// TIA Portal project "Project_Metrou" (V15.1)

(* hardware
DEVICE "S71500/ET200MP station_1"  S7-1500 station
   slot 0: "Rail_0"  Rack  6ES7 590-1***0-0AA0
   slot 1: "PLC_1"  CPU 1513-1 PN  6ES7 513-1AL02-0AB0  V2.6
      slot 3: "CPU display_1"  6ES7591-1AA00-0AA0
*)

// ===== PLC "PLC_1"  CPU 1513-1 PN =====

DATA_BLOCK "Alarme_scara"   // DB1
{ S7_Optimized_Access := 'TRUE' }
VERSION : 0.1
   VAR
      alarme_gather : Word;
      alarme_vect : Array[0..15] of Bool;
   END_VAR
BEGIN
END_DATA_BLOCK

DATA_BLOCK "Avarii"   // DB2
{ S7_Optimized_Access := 'TRUE' }
VERSION : 0.1
   VAR
      esd : Bool;
      esd_btn : Bool;
      reset_esd : Bool;
      avarie_s1 : Bool;
      avarie_s2 : Bool;
      reset_avarii : Bool;
   END_VAR
BEGIN
END_DATA_BLOCK

DATA_BLOCK "Alarme_poarta"   // DB3
{ S7_Optimized_Access := 'TRUE' }
VERSION : 0.1
   VAR
      alarme_gather : Word;
      alarme_vect : Array[0..15] of Bool;
   END_VAR
BEGIN
END_DATA_BLOCK

DATA_BLOCK "Scara1_DB"   // DB4
{ S7_Optimized_Access := 'TRUE' }
VERSION : 0.1
// stored: InstanceOfName Scara
"Scara"
BEGIN
END_DATA_BLOCK

DATA_BLOCK "Scara2_DB"   // DB5
{ S7_Optimized_Access := 'TRUE' }
VERSION : 0.1
// stored: InstanceOfName Scara
"Scara"
BEGIN
END_DATA_BLOCK

DATA_BLOCK "Variabile_scara1"   // DB6
{ S7_Optimized_Access := 'TRUE' }
VERSION : 0.1
   VAR
      curent_stea : Real;
      curent_triunghi : Real;
      senzor_presiune : Bool;
      porniire_stea : Bool;
      pornire_triunghi : Bool;
      start : Bool;
      stop : Bool;
      directie : Bool;
      directie_sus : Bool;
      directie_jos : Bool;
      reseteaza_directia : Bool;
   END_VAR
BEGIN
END_DATA_BLOCK

DATA_BLOCK "Variabile_scara2"   // DB7
{ S7_Optimized_Access := 'TRUE' }
VERSION : 0.1
   VAR
      curent_stea : Real;
      curent_triunghi : Real;
      senzor_presiune : Bool;
      porniire_stea : Bool;
      pornire_triunghi : Bool;
      start : Bool;
      stop : Bool;
      directie : Bool;
      directie_sus : Bool;
      directie_jos : Bool;
      reseteaza_directia : Bool;
   END_VAR
BEGIN
END_DATA_BLOCK

// folder: System blocks/Program resources

DATA_BLOCK "reset_esd"   // DB8
{ S7_Optimized_Access := 'TRUE' }
AUTHOR : Simatic
FAMILY : IEC
NAME : IEC_TMR
VERSION : 1.0
// stored: InstanceOfName IEC_TIMER
"IEC_TIMER"
BEGIN
END_DATA_BLOCK

// folder: (top level)

FUNCTION_BLOCK "Scara"   // FB1, LAD
{ S7_Optimized_Access := 'TRUE' }
VERSION : 0.1
   VAR_INPUT
      esd : Bool;
      curent_stea : Real;
      curent_triunghi : Real;
      senzor_presiune : Bool;
      avarie_scara : Bool;
   END_VAR
   VAR_OUTPUT
      stea : Bool;
      triunghi : Bool;
      directie_selectata : Bool;
   END_VAR
   VAR_IN_OUT
      reseteaza_directia : Bool;
      stop : Bool;
      start : Bool;
      directie_sus : Bool;
      directie_jos : Bool;
   END_VAR
   VAR
      pornire_stea : Bool;
      pornire_triunghi : Bool;
      permisiune_pornire : Bool;
      permisie_repornire : Bool;
      timer_stop : TON_TIME;
      Motor : "Motor";
   END_VAR
BEGIN

REGION Network 1: da permisiuneade pornire la scara
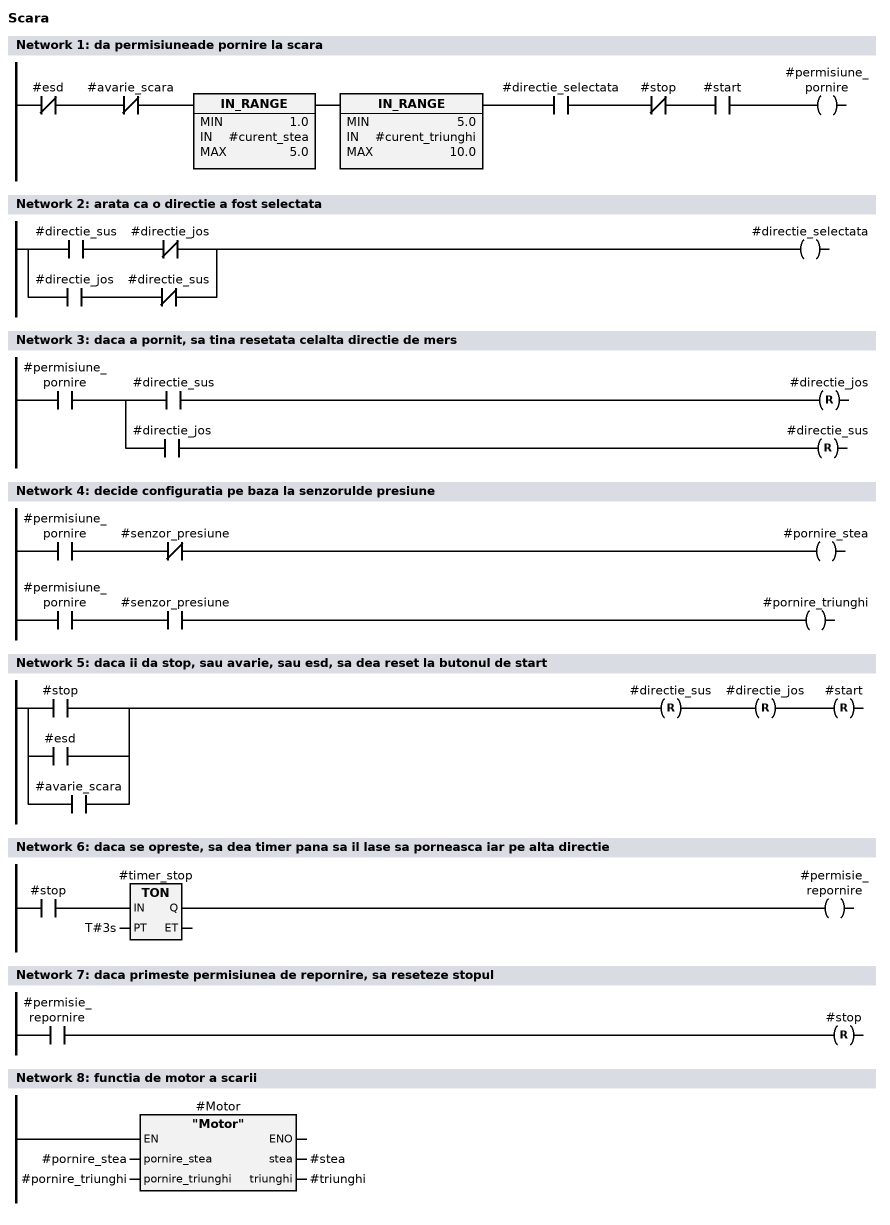
   RUNG wire#powerrail
      I_Contact( #esd )
      I_Contact( #avarie_scara )
      { S7_Templates := "SrcType := Real" } InRange(min := 1.0, in := #curent_stea, max := 5.0)
      { S7_Templates := "SrcType := Real" } InRange(min := 5.0, in := #curent_triunghi, max := 10.0)
      Contact( #directie_selectata )
      I_Contact( #stop )
      Contact( #start )
      Coil( #permisiune_pornire )
   END_RUNG
   // the same network as SCL:
   #permisiune_pornire := NOT #esd AND NOT #avarie_scara AND (1.0 <= #curent_stea) AND (#curent_stea <= 5.0) AND (5.0 <= #curent_triunghi) AND (#curent_triunghi <= 10.0) AND #directie_selectata AND NOT #stop AND #start;
END_REGION

REGION Network 2: arata ca o directie a fost selectata
   RUNG wire#powerrail
      Contact( #directie_sus )
      I_Contact( #directie_jos )
      wire#w1
      Coil( #directie_selectata )
   END_RUNG
   RUNG wire#powerrail
      Contact( #directie_jos )
      I_Contact( #directie_sus )
   END_RUNG wire#w1
   // the same network as SCL:
   #directie_selectata := (#directie_sus AND NOT #directie_jos) OR (#directie_jos AND NOT #directie_sus);
END_REGION

REGION Network 3: daca a pornit, sa tina resetata celalta directie de mers
   RUNG wire#powerrail
      Contact( #permisiune_pornire )
      wire#w1
      Contact( #directie_sus )
      R_Coil( #directie_jos )
   END_RUNG
   RUNG wire#w1
      Contact( #directie_jos )
      R_Coil( #directie_sus )
   END_RUNG
   // the same network as SCL:
   IF #permisiune_pornire AND #directie_sus THEN #directie_jos := FALSE; END_IF;
   IF #permisiune_pornire AND #directie_jos THEN #directie_sus := FALSE; END_IF;
END_REGION

REGION Network 4: decide configuratia pe baza la senzorulde presiune
   RUNG wire#powerrail
      Contact( #permisiune_pornire )
      I_Contact( #senzor_presiune )
      Coil( #pornire_stea )
   END_RUNG
   RUNG wire#powerrail
      Contact( #permisiune_pornire )
      Contact( #senzor_presiune )
      Coil( #pornire_triunghi )
   END_RUNG
   // the same network as SCL:
   #pornire_stea := #permisiune_pornire AND NOT #senzor_presiune;
   #pornire_triunghi := #permisiune_pornire AND #senzor_presiune;
END_REGION

REGION Network 5: daca ii da stop, sau avarie, sau esd, sa dea reset la butonul de start
   RUNG wire#powerrail
      Contact( #stop )
      wire#w1
      R_Coil( #directie_sus )
      R_Coil( #directie_jos )
      R_Coil( #start )
   END_RUNG
   RUNG wire#powerrail
      Contact( #esd )
   END_RUNG wire#w1
   RUNG wire#powerrail
      Contact( #avarie_scara )
   END_RUNG wire#w1
   // the same network as SCL:
   IF #stop OR #esd OR #avarie_scara THEN
       #directie_sus := FALSE;
       #directie_jos := FALSE;
       #start := FALSE;
   END_IF;
END_REGION

REGION Network 6: daca se opreste, sa dea timer pana sa il lase sa porneasca iar pe alta directie
   #timer_stop(IN := #stop, PT := T#3s);   // TON
   #permisie_repornire := #timer_stop.Q;
END_REGION

REGION Network 7: daca primeste permisiunea de repornire, sa reseteze stopul
   RUNG wire#powerrail
      Contact( #permisie_repornire )
      R_Coil( #stop )
   END_RUNG
   // the same network as SCL:
   IF #permisie_repornire THEN #stop := FALSE; END_IF;
END_REGION

REGION Network 8: functia de motor a scarii
   RUNG wire#powerrail
      #Motor(pornire_stea := #pornire_stea, pornire_triunghi := #pornire_triunghi, stea => #stea, triunghi => #triunghi)
   END_RUNG
   // the same network as SCL:
   #Motor(pornire_stea := #pornire_stea,   // "Motor"
          pornire_triunghi := #pornire_triunghi,
          stea => #stea,
          triunghi => #triunghi);
END_REGION
END_FUNCTION_BLOCK

FUNCTION_BLOCK "Motor"   // FB2, LAD
{ S7_Optimized_Access := 'TRUE' }
VERSION : 0.1
   VAR_INPUT
      pornire_stea : Bool;
      pornire_triunghi : Bool;
   END_VAR
   VAR_OUTPUT
      stea : Bool;
      triunghi : Bool;
   END_VAR
BEGIN

REGION Network 1: daca primeste plecare pe stea, sa o activeze
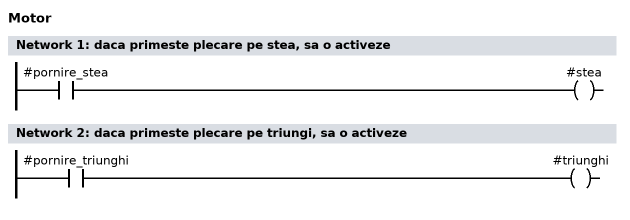
   RUNG wire#powerrail
      Contact( #pornire_stea )
      Coil( #stea )
   END_RUNG
   // the same network as SCL:
   #stea := #pornire_stea;
END_REGION

REGION Network 2: daca primeste plecare pe triungi, sa o activeze
   RUNG wire#powerrail
      Contact( #pornire_triunghi )
      Coil( #triunghi )
   END_RUNG
   // the same network as SCL:
   #triunghi := #pornire_triunghi;
END_REGION
END_FUNCTION_BLOCK

ORGANIZATION_BLOCK "Main"   // OB1, LAD, ProgramCycle
TITLE = "Main Program Sweep (Cycle)"
{ S7_Optimized_Access := 'TRUE' }
VERSION : 0.1
   VAR_INPUT
      Initial_Call : Bool;   // Initial call of this OB
      Remanence : Bool;   // =True, if remanent data are available
   END_VAR
   VAR_TEMP   // added for the SCL form of the ladder/FBD networks
      _w1 : Bool;
      _w2 : Bool;
      _w3 : Bool;
      _w4 : Bool;
      _w5 : Bool;
      _w6 : Bool;
   END_VAR
BEGIN

REGION Network 1: scara 1
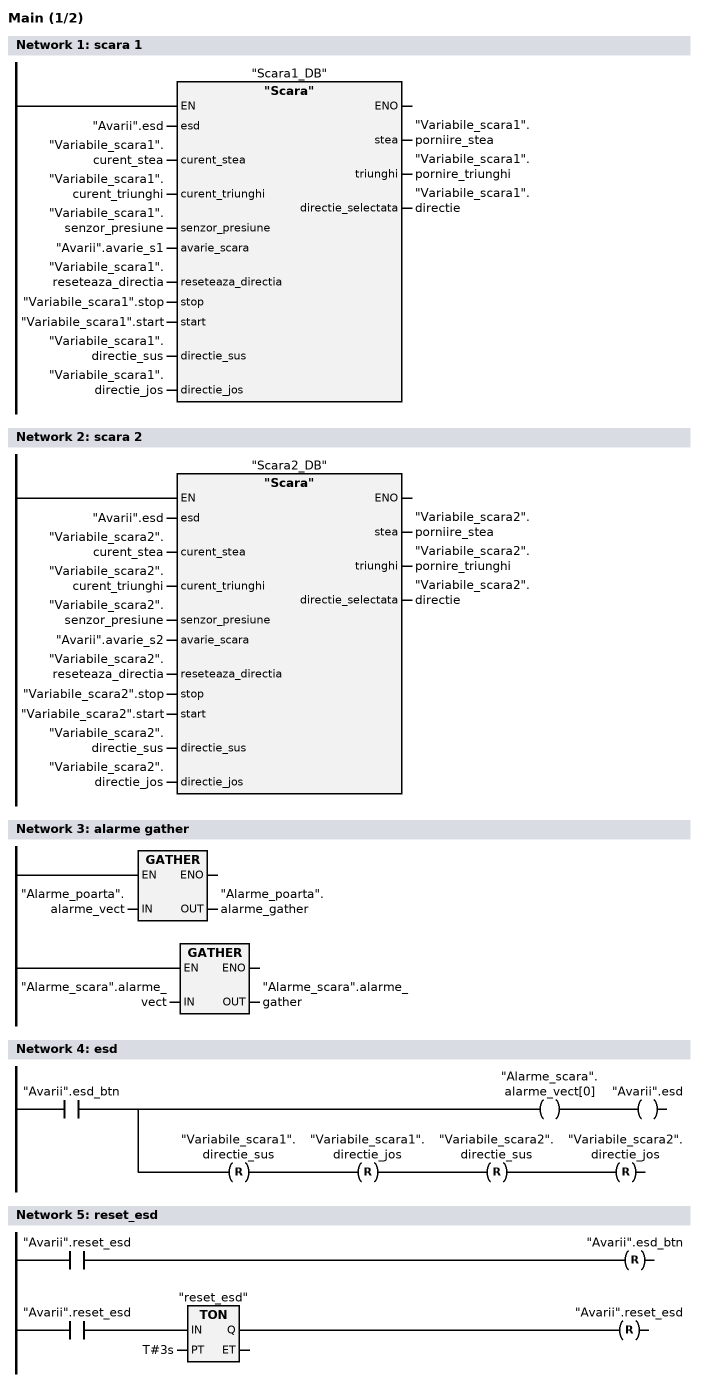
   RUNG wire#powerrail
      "Scara1_DB"(esd := "Avarii".esd, curent_stea := "Variabile_scara1".curent_stea, curent_triunghi := "Variabile_scara1".curent_triunghi, senzor_presiune := "Variabile_scara1".senzor_presiune, avarie_scara := "Avarii".avarie_s1, reseteaza_directia := "Variabile_scara1".reseteaza_directia, stop := "Variabile_scara1".stop, start := "Variabile_scara1".start, directie_sus := "Variabile_scara1".directie_sus, directie_jos := "Variabile_scara1".directie_jos, stea => "Variabile_scara1".porniire_stea, triunghi => "Variabile_scara1".pornire_triunghi, directie_selectata => "Variabile_scara1".directie)
   END_RUNG
   // the same network as SCL:
   "Scara1_DB"(esd := "Avarii".esd,   // "Scara"
               curent_stea := "Variabile_scara1".curent_stea,
               curent_triunghi := "Variabile_scara1".curent_triunghi,
               senzor_presiune := "Variabile_scara1".senzor_presiune,
               avarie_scara := "Avarii".avarie_s1,
               reseteaza_directia := "Variabile_scara1".reseteaza_directia,
               stop := "Variabile_scara1".stop,
               start := "Variabile_scara1".start,
               directie_sus := "Variabile_scara1".directie_sus,
               directie_jos := "Variabile_scara1".directie_jos,
               stea => "Variabile_scara1".porniire_stea,
               triunghi => "Variabile_scara1".pornire_triunghi,
               directie_selectata => "Variabile_scara1".directie);
END_REGION

REGION Network 2: scara 2
   RUNG wire#powerrail
      "Scara2_DB"(esd := "Avarii".esd, curent_stea := "Variabile_scara2".curent_stea, curent_triunghi := "Variabile_scara2".curent_triunghi, senzor_presiune := "Variabile_scara2".senzor_presiune, avarie_scara := "Avarii".avarie_s2, reseteaza_directia := "Variabile_scara2".reseteaza_directia, stop := "Variabile_scara2".stop, start := "Variabile_scara2".start, directie_sus := "Variabile_scara2".directie_sus, directie_jos := "Variabile_scara2".directie_jos, stea => "Variabile_scara2".porniire_stea, triunghi => "Variabile_scara2".pornire_triunghi, directie_selectata => "Variabile_scara2".directie)
   END_RUNG
   // the same network as SCL:
   "Scara2_DB"(esd := "Avarii".esd,   // "Scara"
               curent_stea := "Variabile_scara2".curent_stea,
               curent_triunghi := "Variabile_scara2".curent_triunghi,
               senzor_presiune := "Variabile_scara2".senzor_presiune,
               avarie_scara := "Avarii".avarie_s2,
               reseteaza_directia := "Variabile_scara2".reseteaza_directia,
               stop := "Variabile_scara2".stop,
               start := "Variabile_scara2".start,
               directie_sus := "Variabile_scara2".directie_sus,
               directie_jos := "Variabile_scara2".directie_jos,
               stea => "Variabile_scara2".porniire_stea,
               triunghi => "Variabile_scara2".pornire_triunghi,
               directie_selectata => "Variabile_scara2".directie);
END_REGION

REGION Network 3: alarme gather
   GATHER(IN := "Alarme_poarta".alarme_vect, OUT => "Alarme_poarta".alarme_gather);
   GATHER(IN := "Alarme_scara".alarme_vect, OUT => "Alarme_scara".alarme_gather);
END_REGION

REGION Network 4: esd
   RUNG wire#powerrail
      Contact( "Avarii".esd_btn )
      wire#w1
      Coil( "Alarme_scara".alarme_vect[0] )
      Coil( "Avarii".esd )
   END_RUNG
   RUNG wire#w1
      R_Coil( "Variabile_scara1".directie_sus )
      R_Coil( "Variabile_scara1".directie_jos )
      R_Coil( "Variabile_scara2".directie_sus )
      R_Coil( "Variabile_scara2".directie_jos )
   END_RUNG
   // the same network as SCL:
   "Alarme_scara".alarme_vect[0] := "Avarii".esd_btn;
   "Avarii".esd := "Avarii".esd_btn;
   IF "Avarii".esd_btn THEN
       "Variabile_scara1".directie_sus := FALSE;
       "Variabile_scara1".directie_jos := FALSE;
       "Variabile_scara2".directie_sus := FALSE;
       "Variabile_scara2".directie_jos := FALSE;
   END_IF;
END_REGION

REGION Network 5: reset_esd
   IF "Avarii".reset_esd THEN "Avarii".esd_btn := FALSE; END_IF;
   "reset_esd".TON(IN := "Avarii".reset_esd, PT := T#3s);
   IF "reset_esd".Q THEN "Avarii".reset_esd := FALSE; END_IF;
END_REGION

REGION Network 6: avarii pe scari, cu alarme pt hmi
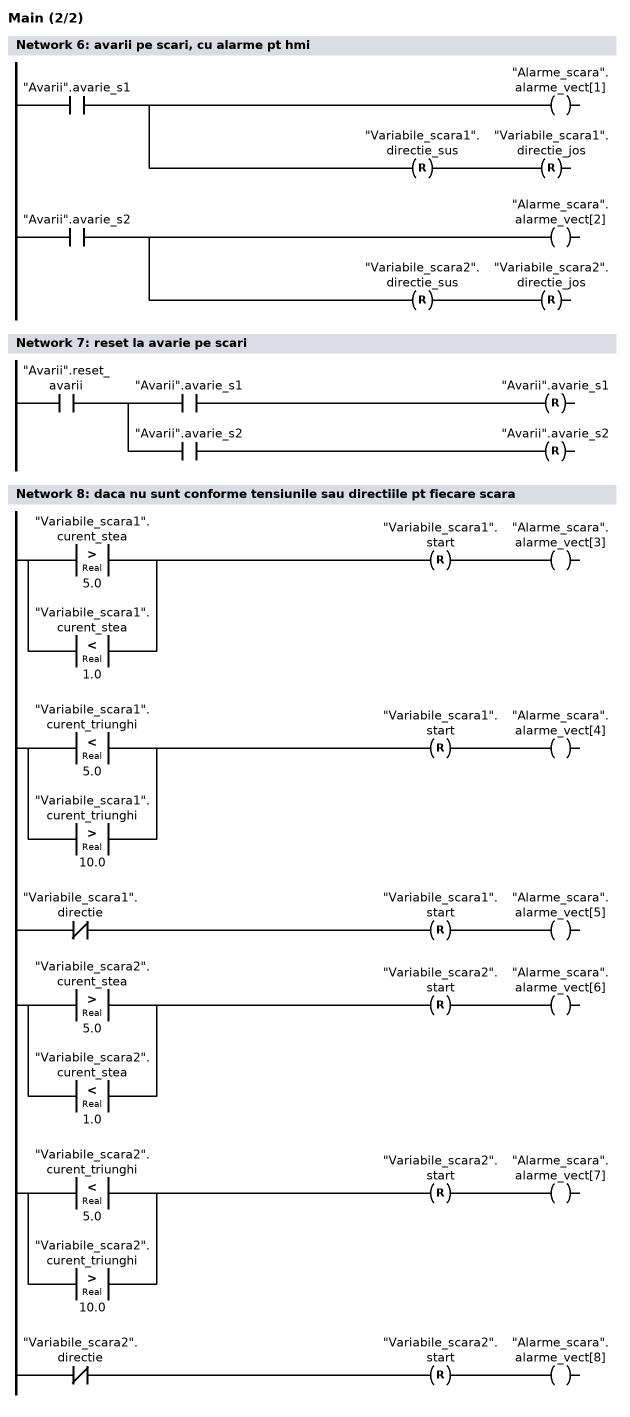
   RUNG wire#powerrail
      Contact( "Avarii".avarie_s1 )
      wire#w1
      Coil( "Alarme_scara".alarme_vect[1] )
   END_RUNG
   RUNG wire#w1
      R_Coil( "Variabile_scara1".directie_sus )
      R_Coil( "Variabile_scara1".directie_jos )
   END_RUNG
   RUNG wire#powerrail
      Contact( "Avarii".avarie_s2 )
      wire#w2
      Coil( "Alarme_scara".alarme_vect[2] )
   END_RUNG
   RUNG wire#w2
      R_Coil( "Variabile_scara2".directie_sus )
      R_Coil( "Variabile_scara2".directie_jos )
   END_RUNG
   // the same network as SCL:
   "Alarme_scara".alarme_vect[1] := "Avarii".avarie_s1;
   IF "Avarii".avarie_s1 THEN
       "Variabile_scara1".directie_sus := FALSE;
       "Variabile_scara1".directie_jos := FALSE;
   END_IF;
   "Alarme_scara".alarme_vect[2] := "Avarii".avarie_s2;
   IF "Avarii".avarie_s2 THEN
       "Variabile_scara2".directie_sus := FALSE;
       "Variabile_scara2".directie_jos := FALSE;
   END_IF;
END_REGION

REGION Network 7: reset la avarie pe scari
   RUNG wire#powerrail
      Contact( "Avarii".reset_avarii )
      wire#w1
      Contact( "Avarii".avarie_s1 )
      R_Coil( "Avarii".avarie_s1 )
   END_RUNG
   RUNG wire#w1
      Contact( "Avarii".avarie_s2 )
      R_Coil( "Avarii".avarie_s2 )
   END_RUNG
   // the same network as SCL:
   IF "Avarii".reset_avarii AND "Avarii".avarie_s1 THEN "Avarii".avarie_s1 := FALSE; END_IF;
   IF "Avarii".reset_avarii AND "Avarii".avarie_s2 THEN "Avarii".avarie_s2 := FALSE; END_IF;
END_REGION

REGION Network 8: daca nu sunt conforme tensiunile sau directiile pt fiecare scara
   RUNG wire#powerrail
      { S7_Templates := "SrcType := Real" } GT_Contact(in1 := "Variabile_scara1".curent_stea, in2 := 5.0)
      wire#w1
      R_Coil( "Variabile_scara1".start )
      Coil( "Alarme_scara".alarme_vect[3] )
   END_RUNG
   RUNG wire#powerrail
      { S7_Templates := "SrcType := Real" } LT_Contact(in1 := "Variabile_scara1".curent_stea, in2 := 1.0)
   END_RUNG wire#w1
   RUNG wire#powerrail
      { S7_Templates := "SrcType := Real" } LT_Contact(in1 := "Variabile_scara1".curent_triunghi, in2 := 5.0)
      wire#w2
      R_Coil( "Variabile_scara1".start )
      Coil( "Alarme_scara".alarme_vect[4] )
   END_RUNG
   RUNG wire#powerrail
      { S7_Templates := "SrcType := Real" } GT_Contact(in1 := "Variabile_scara1".curent_triunghi, in2 := 10.0)
   END_RUNG wire#w2
   RUNG wire#powerrail
      I_Contact( "Variabile_scara1".directie )
      R_Coil( "Variabile_scara1".start )
      Coil( "Alarme_scara".alarme_vect[5] )
   END_RUNG
   RUNG wire#powerrail
      { S7_Templates := "SrcType := Real" } GT_Contact(in1 := "Variabile_scara2".curent_stea, in2 := 5.0)
      wire#w3
      R_Coil( "Variabile_scara2".start )
      Coil( "Alarme_scara".alarme_vect[6] )
   END_RUNG
   RUNG wire#powerrail
      { S7_Templates := "SrcType := Real" } LT_Contact(in1 := "Variabile_scara2".curent_stea, in2 := 1.0)
   END_RUNG wire#w3
   RUNG wire#powerrail
      { S7_Templates := "SrcType := Real" } LT_Contact(in1 := "Variabile_scara2".curent_triunghi, in2 := 5.0)
      wire#w4
      R_Coil( "Variabile_scara2".start )
      Coil( "Alarme_scara".alarme_vect[7] )
   END_RUNG
   RUNG wire#powerrail
      { S7_Templates := "SrcType := Real" } GT_Contact(in1 := "Variabile_scara2".curent_triunghi, in2 := 10.0)
   END_RUNG wire#w4
   RUNG wire#powerrail
      I_Contact( "Variabile_scara2".directie )
      R_Coil( "Variabile_scara2".start )
      Coil( "Alarme_scara".alarme_vect[8] )
   END_RUNG
   // the same network as SCL:
   #_w1 := ("Variabile_scara1".curent_stea > 5.0) OR ("Variabile_scara1".curent_stea < 1.0);
   IF #_w1 THEN "Variabile_scara1".start := FALSE; END_IF;
   "Alarme_scara".alarme_vect[3] := #_w1;
   #_w2 := ("Variabile_scara1".curent_triunghi < 5.0) OR ("Variabile_scara1".curent_triunghi > 10.0);
   IF #_w2 THEN "Variabile_scara1".start := FALSE; END_IF;
   "Alarme_scara".alarme_vect[4] := #_w2;
   #_w3 := NOT "Variabile_scara1".directie;
   IF #_w3 THEN "Variabile_scara1".start := FALSE; END_IF;
   "Alarme_scara".alarme_vect[5] := #_w3;
   #_w4 := ("Variabile_scara2".curent_stea > 5.0) OR ("Variabile_scara2".curent_stea < 1.0);
   IF #_w4 THEN "Variabile_scara2".start := FALSE; END_IF;
   "Alarme_scara".alarme_vect[6] := #_w4;
   #_w5 := ("Variabile_scara2".curent_triunghi < 5.0) OR ("Variabile_scara2".curent_triunghi > 10.0);
   IF #_w5 THEN "Variabile_scara2".start := FALSE; END_IF;
   "Alarme_scara".alarme_vect[7] := #_w5;
   #_w6 := NOT "Variabile_scara2".directie;
   IF #_w6 THEN "Variabile_scara2".start := FALSE; END_IF;
   "Alarme_scara".alarme_vect[8] := #_w6;
END_REGION
END_ORGANIZATION_BLOCK